FUNCTION_BLOCK FB_EventHold
VAR_INPUT
	bEvent		:BOOL;
END_VAR
VAR_OUTPUT
	bEventHold	:BOOL;
END_VAR
VAR
	osTrig		:R_TRIG;
	srEvent		:SR;
	tonHold		:TON;
END_VAR


// One shot trigger for event
osTrig(CLK:= bEvent, Q=> );

// Remember that event has been activated, and hold it untill reset
srEvent(
	SET1:= osTrig.Q, 
	RESET:= tonHold.Q, Q1=> );

// Reset after xx MS
tonHold(IN:= srEvent.Q1, PT:= T#500MS, Q=> , ET=> );

// Set Event Hold
bEventHold := srEvent.Q1;

END_FUNCTION_BLOCK

(* stored: Version 1.1.0.1, ProductVersion 3.1.4024.12
   POU FB_EventHold: Id {3e5acfe3-af83-49c0-9dd9-63ecf11498d6}, SpecialFunc None *)
